// TwinCAT 3 PLC project PRG_B_MachineControl
// Title: B_MachineControl
// Company: RafalOS
// Author: Rafał Osajda
// ProjectVersion: 0.0.0.37
// ProgramVersion: 3.1.4024.0
// libraries:
//   B_Base, * (RafalOS)
//   B_IO, * (RafalOS)
//   B_StatesAndModes, * (RafalOS)
//   Tc2_Standard, * (Beckhoff Automation GmbH)
//   Tc2_System, * (Beckhoff Automation GmbH)
//   Tc3_Module, * (Beckhoff Automation GmbH)
// project tree:
//   / PlcTask.TcTTO (not stored)
//   POUs Compilation/ PRG_Compilation.TcPOU (not stored)
//   POUs/01_MachineControl/ FB_MCMachineControl.TcPOU, ITF_MCMachineControl.TcIO (not stored), ITF_MCMachineControl_HMI_Connector.TcIO, ITF_MCMachineControl_HMI_Init.TcIO, ITF_MCMachineControlConfigure.TcIO, ITF_MCRequiredChange.TcIO (not stored), ST_MCElementListWithParameter.TcDUT, ST_MCRequestChangeMode.TcDUT, ST_MCRequestChangeState.TcDUT (not stored)
//   POUs/02_MachineConfigure/ FB_MCMachineConfigure.TcPOU, ITF_MCConfiguration.TcIO, ITF_MCMachineConfigure.TcIO (not stored)
//   POUs/03_RequiredChange/ FB_MCRequiredChange.TcPOU

// ---- POUs/01_MachineControl/ST_MCElementListWithParameter.TcDUT
TYPE ST_MCElementListWithParameter :
STRUCT
	arrNames 			: ARRAY  [1..GVL_BaseConstans.MAX_NUMBER_OF_ALL_ITEM] OF WSTRING;
	arrID				: ARRAY  [1..GVL_BaseConstans.MAX_NUMBER_OF_ALL_ITEM] OF UINT;
	iNumber				: INT;	//liczba elementów z parametrami
END_STRUCT
END_TYPE

// ---- POUs/01_MachineControl/ST_MCRequestChangeMode.TcDUT
TYPE ST_MCRequestChangeMode :
STRUCT

END_STRUCT
END_TYPE

// ---- POUs/01_MachineControl/ITF_MCMachineControl_HMI_Connector.TcIO
INTERFACE ITF_MCMachineControl_HMI_Connector EXTENDS ITF_BaseTopElement_HMI_Connector

(*			
	RafalOS
	Rafał Osajda		25.11.2025		TC 4024.66
	Zwraca aktualny tryb
*)
METHOD PUBLIC GetActiveMode : E_BaseMachineMode
VAR_INPUT
END_VAR
END_METHOD

METHOD PUBLIC GetActiveModeName : ST_BaseLabel
VAR_INPUT
END_VAR
END_METHOD

(*			
	RafalOS
	Rafał Osajda		25.11.2025		TC 4024.66
	Zwraca aktualny stan
*)
METHOD PUBLIC GetActiveState : E_BaseMachineState
VAR_INPUT
END_VAR
END_METHOD

METHOD PUBLIC GetActiveStateName : ST_BaseLabel
VAR_INPUT
END_VAR
END_METHOD

(*			
	RafalOS
	Rafał Osajda		17.12.2025		TC 4024.66
	Pobiera listę elementów które posiadaja parametr i 
	przypisuje ja do zadanej struktury i zwraca true jak się uda
*)
METHOD GetElementNamesWithParameter : BOOL
VAR_INPUT
	stDane			: REFERENCE TO ST_MCElementListWithParameter;
END_VAR
END_METHOD

METHOD PUBLIC GetModeName : ST_BaseLabel
VAR_INPUT
	iNumber		: INT;
END_VAR
END_METHOD

METHOD PUBLIC GetStateName : ST_BaseLabel
VAR_INPUT
	iNumber		: INT;
END_VAR
END_METHOD

METHOD GetStateTimeForCurrentMode : LTIME
VAR_INPUT
	iNumber			: INT;
END_VAR
END_METHOD

METHOD GetStateTimeForMode : LTIME
VAR_INPUT
	iMode			: INT;
	iState			: INT;
END_VAR
END_METHOD

METHOD PUBLIC GetTimeWorkForMode : LTIME
VAR_INPUT
	iMode	: INT;
END_VAR
END_METHOD

(*			
	RafalOS
	Rafał Osajda		25.11.2025		TC 4024.66
	Zwraca całkowity czas pracy maszyny
*)
METHOD PUBLIC GetTotalWorkTime : LTIME
VAR_INPUT
END_VAR
END_METHOD

(*			
	RafalOS
	Rafał Osajda		25.11.2025		TC 4024.66
	Zwraca czy zmiana trybu sie skoćńzyła
*)
METHOD PUBLIC IsChangeModeDone : BOOL
VAR_INPUT
END_VAR
END_METHOD

(*			
	RafalOS
	Rafał Osajda		25.11.2025		TC 4024.66
	Zwraca czy tryb o podanym numerze jest włączony
*)
METHOD IsModeEnabled : BOOL
VAR_INPUT
	iMode 	: INT;
END_VAR
END_METHOD

(*			
	RafalOS
	Rafał Osajda		24.11.2025		TC 4024.66
	Informacja czy dany stan jest aktywny w aktualnym trybie trybie
*)
METHOD PUBLIC IsStateActiveInCurrentMode : BOOL
VAR_INPUT
END_VAR
END_METHOD

(*			
	RafalOS
	Rafał Osajda		25.11.2025		TC 4024.66
	Informacja czy zadany stan jest stanem aktualnym
*)
METHOD PUBLIC IsStateIsActual : BOOL
VAR_INPUT
	iTestState	: INT;
END_VAR
END_METHOD

METHOD PUBLIC SetCmdChangeMode
VAR_INPUT
	eCmdNumber		: E_SaMCommandChangeMode;
END_VAR
END_METHOD

METHOD PUBLIC SetCmdChangeState
VAR_INPUT
	eCmdNumber		: E_SaMCommandChangeState;
END_VAR
END_METHOD

END_INTERFACE

// ---- POUs/01_MachineControl/ITF_MCMachineControl_HMI_Init.TcIO
INTERFACE ITF_MCMachineControl_HMI_Init EXTENDS ITF_BaseTopElement, ITF_MCMachineControl_HMI_Connector

END_INTERFACE

// ---- POUs/01_MachineControl/ITF_MCMachineControlConfigure.TcIO
(*			
	RafalOS
	Rafał Osajda		29.10.2025		TC 4024.66
	Metody do konfiguracji MAchine control wywoływane z MachineConfigure z pomocą przekazanego ITF
*)
INTERFACE ITF_MCMachineControlConfigure EXTENDS ITF_Base

(*			
	RafalOS
	Rafał Osajda		26.11.2025		TC 4024.66
	Dodawanie szablonu receptury
*)
METHOD PUBLIC AddCreateTemplateFromConfiguration : BOOL
VAR_INPUT
	fbCreateTemplate			: ITF_BaseCreateTemplateOfRecipe;
END_VAR
END_METHOD

(*			
	RafalOS
	Rafał Osajda		13.11.2025		TC 4024.66
	Dodawanie elementów wywoływane z konfiguracji 
*)
METHOD PUBLIC AddElementFromConfiguration : BOOL
VAR_INPUT
	itfElements		: ITF_BaseTopElement;
END_VAR
END_METHOD

(*			
	RafalOS
	Rafał Osajda		13.11.2025		TC 4024.66
	Podpięcie menadżera HMI wywoływane z konfiguracji
*)
METHOD AddHMIManagerFromConfiguration : BOOL
VAR_INPUT
	fbHMIManager			: ITF_BaseGroupElement;
END_VAR
END_METHOD

(*			
	RafalOS
	Rafał Osajda		13.11.2025		TC 4024.66
	Dodanie samego sibie do obsługi w MachineControl
*)
METHOD PUBLIC AddMachineCotrolToYourSelfFromConfiguration : BOOL
VAR_INPUT
END_VAR
END_METHOD

(*			
	RafalOS
	Rafał Osajda		26.11.2025		TC 4024.66
	Dodanie obsługi receptur
*)
METHOD PUBLIC AddModulRecipeFromConfiguration : BOOL
VAR_INPUT
	itfRecipe			: ITF_BaseRecipe;
END_VAR
END_METHOD

(*			
	RafalOS
	Rafał Osajda		13.11.2025		TC 4024.66
	Dodanie modułu sterowania stanami i trybami do machinecontrol z konfiguracji
*)
METHOD PUBLIC AddSaMCotrollerToMachineControlFromConfiguration : BOOL
VAR_INPUT
	itfSaMController			: ITF_SaMController;
END_VAR
END_METHOD

METHOD PUBLIC AddSaMToTopElementFromConfiguration
VAR_INPUT
	itfSaMController			: ITF_SaMController;
END_VAR
END_METHOD

(*			
	RafalOS
	Rafał Osajda		13.11.2025		TC 4024.66
	Wywołanie pierwszego przejścia u wszystkich podzepsołów
*)
METHOD PUBLIC ExecuteFirstCycle : BOOL
VAR_INPUT
END_VAR
END_METHOD

(*			
	RafalOS
	Rafał Osajda		13.11.2025		TC 4024.66
	Zlinkowanie danych wspólnych do dodanych elementów wywoływane z konfiguracji
*)
METHOD PUBLIC LinkCommonDataToAddedElementsFromConfiguration : BOOL
VAR_INPUT
	stCommonData		: REFERENCE TO ST_BaseCommonData;
END_VAR
END_METHOD

(*			
	RafalOS
	Rafał Osajda		13.11.2025		TC 4024.66
	Dodanie głównego komunikatora pomiędzy topelementami do topelementów wywolywane z konfiguracji
*)
METHOD PUBLIC LinkMassangerToaddedTopElementsFromConfiguration : BOOL
VAR_INPUT
	fbCommunicator		: ITF_BaseCommunicator;
END_VAR
END_METHOD

(*			
	RafalOS
	Rafał Osajda		14.11.2025		TC 4024.66
	Podpięcie przyciskow zmiany stanu wywoływane z konfiguracji 
*)
METHOD LinkRequestButtonModeChangeFromConfiguration : BOOL
VAR_INPUT
	iNumberOfRequest			: INT;
	itfRequest					: ITF_MCRequiredChange;
END_VAR
END_METHOD

(*			
	RafalOS
	Rafał Osajda		14.11.2025		TC 4024.66
	Podpięcie przyciskow zmiany trybu i stanu wywoływane z konfiguracji 
*)
METHOD LinkRequestButtonStateChangeFromConfiguration : BOOL
VAR_INPUT
	iNumberOfRequest			: INT;
	itfRequest					: ITF_MCRequiredChange;
END_VAR
END_METHOD

(*			
	RafalOS
	Rafał Osajda		13.11.2025		TC 4024.66
	Podłączenie wsyzstkich zmiennych pochodzących od Programu safety wywoływane w konfiguratorze
*)
METHOD PUBLIC LinkSafetyToaddedElementsFromConfiguration : BOOL
VAR_INPUT
	flSS1				: ITF_BaseFlagGet;
	flSTO				: ITF_BaseFlagGet;
END_VAR
END_METHOD

(*			
	RafalOS
	Rafał Osajda		13.11.2025		TC 4024.66
	Nadanie unikalnych kodów elementom w systemie wywołane z konfiguracji
*)
METHOD PUBLIC SetCodeToAddedElementsFromConfiguration : BOOL
VAR_INPUT
END_VAR
END_METHOD

(*			
	RafalOS
	Rafał Osajda		13.11.2025		TC 4024.66
	Uruchomienie lub wyłączenie obsługi HMI jak jest false fb obsługi nie jest dodawane do MachineControl wywolywane z konfiguracji
*)
METHOD SetEnableHMIServiceFromConfiguration : BOOL
VAR_INPUT
	bValue		: BOOL;
END_VAR
END_METHOD

(*			
	RafalOS
	Rafał Osajda		13.11.2025		TC 4024.66
	Nadaje unikalne ID zgłoszeniom dodanym do elementów w sesyemie wywołane z konfiguracji
*)
METHOD PUBLIC SetIDEventsToAddedElementsFromConfiguration : BOOL
VAR_INPUT
END_VAR
END_METHOD

(*			
	RafalOS
	Rafał Osajda		13.11.2025		TC 4024.66
	Dodanie wszystkim elementom w systemie unikalnego ID
*)
METHOD PUBLIC SetIDToAddedElementsFromConfiguration : BOOL
VAR_INPUT
END_VAR
END_METHOD

(*			
	RafalOS
	Rafał Osajda		14.11.2025		TC 4024.66
	ustawienie trybu poczatkowego wywoływane z konfiguracji
*)
METHOD SetStartModeFromConfiguration : BOOL
VAR_INPUT
	eStartMode				: E_BaseMachineMode;
END_VAR
END_METHOD

END_INTERFACE

// ---- POUs/02_MachineConfigure/ITF_MCConfiguration.TcIO
(*			
	RafalOS
	Rafał Osajda		10.11.2025		TC 4024.66
	Interfejs metod do konfiguracji FB wywoływane z FB_Cofigure
*)
INTERFACE ITF_MCConfiguration

(*			
	RafalOS
	Rafał Osajda		26.11.2025		TC 4024.66
	Dodawanie szablonu receptury
*)
METHOD PUBLIC AddCreateTemplate : BOOL
VAR_INPUT
	itfMachineControl			: ITF_MCMachineControlConfigure;
END_VAR
END_METHOD

(*			
	RafalOS
	Rafał Osajda		13.11.2025		TC 4024.66
	Metoda przeznaczona do dodawania elementów do FB_MachineControl
*)
METHOD PUBLIC AddElements : BOOL
VAR_INPUT
	itfMachineControl			: ITF_MCMachineControlConfigure;
END_VAR
END_METHOD

(*			
	RafalOS
	Rafał Osajda		13.11.2025		TC 4024.66
	Podpięcie menadżera HMI
*)
METHOD AddHMIManager : BOOL
VAR_INPUT
	itfMachineControl			: ITF_MCMachineControlConfigure;
END_VAR
END_METHOD

(*			
	RafalOS
	Rafał Osajda		13.11.2025		TC 4024.66
	Dodanie samego siebie do systemu controli maszyny
*)
METHOD PUBLIC AddMachineCotrolToYourSelf : BOOL
VAR_INPUT
	itfMachineControl			: ITF_MCMachineControlConfigure;
END_VAR
END_METHOD

(*			
	RafalOS
	Rafał Osajda		26.11.2025		TC 4024.66
	Dodanie obsługi receptur
*)
METHOD PUBLIC AddModulRecipe : BOOL
VAR_INPUT
	itfMachineControl			: ITF_MCMachineControlConfigure;
END_VAR
END_METHOD

(*			
	RafalOS
	Rafał Osajda		13.11.2025		TC 4024.66
	Dodanie modułu sterowania stanami i trybami do machinecontrol
*)
METHOD PUBLIC AddSaMCotrollerToMachineControl : BOOL
VAR_INPUT
	itfMachineControl			: ITF_MCMachineControlConfigure;
END_VAR
END_METHOD

METHOD PUBLIC AddSaMToTopElement
VAR_INPUT
	itfMachineControl			: ITF_MCMachineControlConfigure;
END_VAR
END_METHOD

(*			
	RafalOS
	Rafał Osajda		13.11.2025		TC 4024.66
	Zlinkowanie danych wspólnych do dodanych elementów
*)
METHOD PUBLIC LinkCommonDataToAddedElements : BOOL
VAR_INPUT
	itfMachineControl			: ITF_MCMachineControlConfigure;
END_VAR
END_METHOD

(*			
	RafalOS
	Rafał Osajda		13.11.2025		TC 4024.66
	Dodanie głównego komunikatora pomiędzy topelementami do topelementów
*)
METHOD PUBLIC LinkMassangerToaddedTopElements : BOOL
VAR_INPUT
	itfMachineControl			: ITF_MCMachineControlConfigure;
END_VAR
END_METHOD

(*			
	RafalOS
	Rafał Osajda		14.11.2025		TC 4024.66
	Podpięcie przyciskow zmiany trybu i stanu
*)
METHOD LinkRequestButtonChange : BOOL
VAR_INPUT
	itfMachineControl			: ITF_MCMachineControlConfigure;
END_VAR
END_METHOD

(*			
	RafalOS
	Rafał Osajda		13.11.2025		TC 4024.66
	Podłączenie wsyzstkich zmiennych pochodzących od Programu safety 
*)
METHOD PUBLIC LinkSafetyToaddedElements : BOOL
VAR_INPUT
	itfMachineControl			: ITF_MCMachineControlConfigure;
END_VAR
END_METHOD

(*			
	RafalOS
	Rafał Osajda		13.11.2025		TC 4024.66
	Nadanie unikalnych kodów elementom w systemie
*)
METHOD PUBLIC SetCodeToAddedElements : BOOL
VAR_INPUT
	itfMachineControl			: ITF_MCMachineControlConfigure;
END_VAR
END_METHOD

(*			
	RafalOS
	Rafał Osajda		13.11.2025		TC 4024.66
	Uruchomienie lub wyłączenie obsługi HMI jak jest false fb obsługi nie jest dodawane do MachineControl
*)
METHOD SetEnableHMIService : BOOL
VAR_INPUT
	itfMachineControl			: ITF_MCMachineControlConfigure;
END_VAR
END_METHOD

(*			
	RafalOS
	Rafał Osajda		13.11.2025		TC 4024.66
	Nadaje unikalne ID zgłoszeniom dodanym do elementów w sesyemie
*)
METHOD PUBLIC SetIDEventsToAddedElements : BOOL
VAR_INPUT
	itfMachineControl			: ITF_MCMachineControlConfigure;
END_VAR
END_METHOD

(*			
	RafalOS
	Rafał Osajda		13.11.2025		TC 4024.66
	Dodanie wszystkim elementom w systemie unikalnego ID
*)
METHOD PUBLIC SetIDToAddedElements : BOOL
VAR_INPUT
	itfMachineControl			: ITF_MCMachineControlConfigure;
END_VAR
END_METHOD

(*			
	RafalOS
	Rafał Osajda		14.11.2025		TC 4024.66
	ustawienie trybu poczatkowego
*)
METHOD SetStartMode : BOOL
VAR_INPUT
	itfMachineControl			: ITF_MCMachineControlConfigure;
END_VAR
END_METHOD

END_INTERFACE

// ---- POUs/01_MachineControl/FB_MCMachineControl.TcPOU
(*			
	RafalOS
	Rafał Osajda		04.11.2025		TC 4024.66
	Główny FB zarządzający pracą maszyny
*)
FUNCTION_BLOCK FB_MCMachineControl EXTENDS FB_BaseTopElement IMPLEMENTS ITF_MCMachineControl, ITF_MCMachineControlConfigure, ITF_MCMachineControl_HMI_Init
VAR
	(*	Inicjalizacja		*)
	bInitializeCycle			: BOOL;
	bInitDone					: BOOL;
	(*	Konfiguracja		*)
	itfMachineConfigure			: ITF_MCMachineConfigure;		//moduł konfiguracji
	bEnableHMIService			: BOOL;
	(*	TopElementy systemu	*)
	arrTopElements					: ARRAY [1..GVL_BaseConstans.MAX_NUMBER_OF_TOP_ELEMENT] OF ITF_BaseTopElement;
	uiNumberOfAddedTopElement		: UINT := 0;//przy dodawaniu element 0 to system 
	uiNumberOfAllAddedElements		: UINT;		//liczba elementow które są na maszynie 
	(*	Master komunikatora dla top elementów maszyny	*)
	fbMasterCommunicator			: FB_BaseCommunicator;
	(*	Zarządzenia stanami i trybami pracy	*)
	itfSaMController				: ITF_SaMController;
	(*	Stany i Tryby	*)
	arrRequestChangeState			: ARRAY [1..GVL_SaMConstans.NUMBER_OF_COMMAND_CHANGE_STATES] OF ITF_MCRequiredChange;
	arrRequestChangeMode			: ARRAY [1..GVL_SaMConstans.NUMBER_OF_COMMAND_CHANGE_MODES] OF ITF_MCRequiredChange;
	(*	Tablica informacyjna czy praca w stanie aktywnym zakończona	*)
	arrTopElementWorkFinishedInState	: ARRAY [1..GVL_SaMConstans.NUMBER_OF_STATES] OF BOOL;
	(*	Receptury	*)
	itfRecipe						: ITF_BaseRecipe;
	bWorkWithRecipe					: BOOL;
END_VAR
VAR PERSISTENT
	ltWorkTime						: LTIME;				//czas pracy w danym stanie - trybie
END_VAR

IF (NOT THIS^.bInitializeCycle) THEN
	THIS^.bInitializeCycle		:= TRUE;
	THIS^.bInitDone				:= THIS^.InitializeCycle ();
ELSIF (THIS^.bInitDone) THEN
	THIS^.ExecuteCycle ();
END_IF

(*			
	RafalOS
	Rafał Osajda		26.11.2025		TC 4024.66
	Dodawanie szablonu receptury
*)
METHOD PUBLIC AddCreateTemplateFromConfiguration : BOOL
VAR_INPUT
	fbCreateTemplate			: ITF_BaseCreateTemplateOfRecipe;
END_VAR
THIS^.itfRecipe.AddITFToCreateTemplate (fbToCtreateTemplate := fbCreateTemplate);
END_METHOD

(*			
	RafalOS
	Rafał Osajda		13.11.2025		TC 4024.66
	Dodawanie elementów wywoływane z konfiguracji 
*)
METHOD PUBLIC AddElementFromConfiguration : BOOL
VAR_INPUT
	itfElements		: ITF_BaseTopElement;
END_VAR
IF (THIS^.uiNumberOfAddedTopElement + 1 <= GVL_BaseConstans.MAX_NUMBER_OF_TOP_ELEMENT) THEN
	THIS^.uiNumberOfAddedTopElement := THIS^.uiNumberOfAddedTopElement + 1;
	THIS^.arrTopElements [THIS^.uiNumberOfAddedTopElement] := itfElements;

	AddElementFromConfiguration := TRUE;
END_IF
END_METHOD

(*			
	RafalOS
	Rafał Osajda		13.11.2025		TC 4024.66
	Podpięcie menadżera HMI wywoływane z konfiguracji
*)
METHOD AddHMIManagerFromConfiguration : BOOL
VAR_INPUT
	fbHMIManager			: ITF_BaseGroupElement;
END_VAR
IF (THIS^.bEnableHMIService) THEN
	THIS^.AddControlElement (itfControlElement := fbHMIManager);
	
END_IF
END_METHOD

(*			
	RafalOS
	Rafał Osajda		13.11.2025		TC 4024.66
	Dodanie samego sibie do obsługi w MachineControl
*)
METHOD PUBLIC AddMachineCotrolToYourSelfFromConfiguration : BOOL
VAR_INPUT
END_VAR
THIS^.uiNumberOfAddedTopElement := THIS^.uiNumberOfAddedTopElement + 1;
THIS^.arrTopElements [THIS^.uiNumberOfAddedTopElement]	:= THIS^;
END_METHOD

(*			
	RafalOS
	Rafał Osajda		29.10.2025		TC 4024.66
	Dodawanie intefejsu konfiguracji
*)
METHOD PUBLIC AddModulConfigure : BOOL
VAR_INPUT
	fbMachineConfigure			: ITF_MCMachineConfigure;
END_VAR
THIS^.itfMachineConfigure		:= fbMachineConfigure;
END_METHOD

(*			
	RafalOS
	Rafał Osajda		26.11.2025		TC 4024.66
	Dodanie obsługi receptur
*)
METHOD PUBLIC AddModulRecipeFromConfiguration : BOOL
VAR_INPUT
	itfRecipe			: ITF_BaseRecipe;
END_VAR
THIS^.itfRecipe := itfRecipe;
END_METHOD

METHOD PUBLIC AddModulSaM : BOOL
VAR_INPUT
	fbSaMController			: ITF_SaMController;
END_VAR
THIS^.itfSaMController		:= fbSaMController;
THIS^.AddControlElement (itfControlElement	:= fbSaMController);
END_METHOD

(*			
	RafalOS
	Rafał Osajda		13.11.2025		TC 4024.66
	Dodanie modułu sterowania stanami i trybami do machinecontrol z konfiguracji
*)
METHOD PUBLIC AddSaMCotrollerToMachineControlFromConfiguration : BOOL
VAR_INPUT
	itfSaMController			: ITF_SaMController;
END_VAR
VAR
	iNumberOfTopElement			: INT;
END_VAR
THIS^.AddControlElement (itfControlElement := itfSaMController);
THIS^.itfSaMController := itfSaMController;
//FOR iNumberOfTopElement := 1 TO TO_INT (THIS^.uiNumberOfAddedTopElement) DO
//	THIS^.arrTopElements [iNumberOfTopElement].LinkSaM (
//		fbSAM := itfSaMController
//	);
//END_FOR
END_METHOD

METHOD PUBLIC AddSaMToTopElementFromConfiguration
VAR_INPUT
	itfSaMController			: ITF_SaMController;
END_VAR

VAR
	iNumberOfTopElement: INT;
END_VAR
FOR iNumberOfTopElement := 1 TO TO_INT (THIS^.uiNumberOfAddedTopElement) DO
	THIS^.arrTopElements [iNumberOfTopElement].LinkSaM (
		fbSAM := itfSaMController
	);
END_FOR
END_METHOD

METHOD PRIVATE ExecuteCycle
VAR_INST
	tonInterval	: TON;
END_VAR
VAR
	iI			: INT;
	tInterval	: TIME := T#100MS;
END_VAR
	(*	Zarządzanie Stanami i Trybami	*)

THIS^.ExecuteCycle_SaM ();

	(*	Obsługa czasu *)

tonInterval (IN := NOT tonInterval.Q, PT := tInterval);
IF (tonInterval.Q) THEN
	THIS^.itfSaMController.IncrementTimeStateAndMode (tInterval := tInterval);
	THIS^.ltWorkTime := THIS^.ltWorkTime + TO_LTIME (tInterval);
END_IF

	(*	Wywołanie metod obsługiwanych co cykl dla każdego elementu	*)

FOR iI := 1 TO TO_INT (THIS^.uiNumberOfAddedTopElement) DO
	THIS^.arrTopElements [iI].ExecuteEveryCycle_Test ();
	THIS^.arrTopElements [iI].ExecuteEveryCycle_Operation ();
	THIS^.arrTopElements [iI].ExecuteEveryCycle_Status ();
	THIS^.arrTopElements [iI].ExecuteEveryCycle_Error ();
	
END_FOR
END_METHOD

METHOD PRIVATE ExecuteCycle_SaM
VAR
	iI					: INT;
	bBlockade			: BOOL;	//polecenie zmiany trybu i nie sprawdzaj czy jest polecenie zmiany stanu
	bTypeStateActive		: BOOL;
	bTopElementStateWorkCompleted	: BOOL;	//praca w trybach aktywnych zakończona
	
END_VAR

	(*	Zarządzanie stanami i trybami pracy 	*)

IF (NOT THIS^.itfSaMController.IsChangeModeBusy () AND NOT THIS^.itfSaMController.IsChangeStateBusy ()) THEN	
	(*	Testowanie czy jest rządzanie zmiany trybu	*)
	FOR iI := 1 TO GVL_SaMConstans.NUMBER_OF_COMMAND_CHANGE_MODES DO 
		IF (THIS^.arrRequestChangeMode [iI] <> 0) THEN
			IF (THIS^.arrRequestChangeMode [iI].Testing ()) THEN
				THIS^.itfSaMController.Execute (iNumberOfCommand := iI, eChangeCategory := E_SaMChangeCategory.eMode);
				bBlockade		:= TRUE;
				EXIT;
			END_IF
		END_IF
	END_FOR	
	
	(*	Testowanie czy jest rządanie zmiany stany	*)
	IF (NOT bBlockade) THEN
		IF (THIS^.itfSaMController.GetMode () <> E_BaseMachineMode.NotAllowed AND
			THIS^.itfSaMController.GetState () = E_BaseMachineState.Undefined) THEN
			
			THIS^.itfSaMController.Execute (
				iNumberOfCommand := E_SaMCommandChangeState.Abort,
				eChangeCategory := E_SaMChangeCategory.eState
			);
			
		ELSE
			
			FOR iI := 1 TO GVL_SaMConstans.NUMBER_OF_COMMAND_CHANGE_STATES DO 
				IF (THIS^.arrRequestChangeState [iI] <> 0) THEN
					IF (THIS^.arrRequestChangeState [iI].Testing ()) THEN
						THIS^.itfSaMController.Execute (
							iNumberOfCommand := iI,
							eChangeCategory := E_SaMChangeCategory.eState
						);
						EXIT;
					END_IF
				END_IF
			END_FOR
			
		END_IF
	END_IF

END_IF

	(*	Obsługa stanów 		*)
//informacja czy jesteśny w stanie aktywnym	
bTypeStateActive	 := SEL (THIS^.itfSaMController.GetState () <> E_BaseMachineState.Undefined,FALSE,THIS^.itfSaMController.IsStateTypeActive ());
IF (THIS^.itfSaMController.IsChangeModeDone () AND THIS^.itfSaMController.IsChangeStateDone ()) THEN
	bTopElementStateWorkCompleted := bTypeStateActive;
	IF (THIS^.itfSaMController.GetState () <> E_BaseMachineState.Undefined) THEN
		FOR iI := 1 TO TO_INT (THIS^.uiNumberOfAddedTopElement) DO
			IF ( (bTypeStateActive AND NOT THIS^.arrTopElementWorkFinishedInState [iI]) OR NOT bTypeStateActive) THEN
				THIS^.arrTopElementWorkFinishedInState [iI]	:= THIS^.itfSaMController.ExecuteTopElementOperationsForCurrentState (itfTopElement := THIS^.arrTopElements [iI]);
				bTopElementStateWorkCompleted			:= bTopElementStateWorkCompleted AND THIS^.arrTopElementWorkFinishedInState [iI];
			END_IF
		END_FOR
	END_IF
END_IF
(*	OPeracja zakonczona wyczysc tablice dla kolejnej zmiany stanow i konczenia pracy	*)
IF (bTopElementStateWorkCompleted) THEN
	MEMSET (
		destAddr							:= ADR (THIS^.arrTopElementWorkFinishedInState),
		fillByte							:= 0,
		n									:= SIZEOF (THIS^.arrTopElementWorkFinishedInState)
	);
	(*	Zmiana stanu na następny wyjście ze stanu aktywnego	*)
	THIS^.itfSaMController.ExitActivState ();
END_IF
END_METHOD

(*			
	RafalOS
	Rafał Osajda		13.11.2025		TC 4024.66
	Wywołanie pierwszego przejścia u wszystkich podzepsołów
*)
METHOD PUBLIC ExecuteFirstCycle : BOOL
VAR_INPUT
END_VAR

VAR
	iNumberOfTopElement: INT;
END_VAR
FOR iNumberOfTopElement := 1 TO TO_INT (THIS^.uiNumberOfAddedTopElement) DO
	THIS^.arrTopElements [iNumberOfTopElement].FirstCycle ();
END_FOR
END_METHOD

(*			
	RafalOS
	Rafał Osajda		25.11.2025		TC 4024.66
	Zwraca aktualny tryb
*)
METHOD PUBLIC GetActiveMode : E_BaseMachineMode
VAR_INPUT
END_VAR
GetActiveMode := THIS^.itfSaMController.GetMode ();
END_METHOD

METHOD PUBLIC GetActiveModeName : ST_BaseLabel
VAR_INPUT
END_VAR
GetActiveModeName := THIS^.itfSaMController.GetActiveModeName ();
END_METHOD

(*			
	RafalOS
	Rafał Osajda		25.11.2025		TC 4024.66
	Zwraca aktualny stan
*)
METHOD PUBLIC GetActiveState : E_BaseMachineState
VAR_INPUT
END_VAR
GetActiveState := THIS^.itfSaMController.GetState ();
END_METHOD

METHOD PUBLIC GetActiveStateName : ST_BaseLabel
VAR_INPUT
END_VAR
GetActiveStateName := THIS^.itfSaMController.GetActiveStateName ();
END_METHOD

METHOD PUBLIC GetCommunicatorITF : ITF_BaseCommunicator
VAR_INPUT
END_VAR
GetCommunicatorITF := THIS^.fbMasterCommunicator;
END_METHOD

(*			
	RafalOS
	Rafał Osajda		17.12.2025		TC 4024.66
	Pobiera listę elementów które posiadaja parametr i 
	przypisuje ja do zadanej struktury i zwraca true jak się uda
*)
METHOD GetElementNamesWithParameter : BOOL
VAR_INPUT
	stDane			: REFERENCE TO ST_MCElementListWithParameter;
END_VAR

VAR
	iI: INT;
END_VAR
FOR iI := 1 TO TO_INT (THIS^.uiNumberOfAddedTopElement) DO
	;
END_FOR
END_METHOD

METHOD PUBLIC GetModeName : ST_BaseLabel
VAR_INPUT
	iNumber		: INT;
END_VAR
GetModeName := THIS^.itfSaMController.GetModeName (iNumber := iNumber);
END_METHOD

METHOD PUBLIC GetStateName : ST_BaseLabel
VAR_INPUT
	iNumber		: INT;
END_VAR
GetStateName := THIS^.itfSaMController.GetStateName (iNumber := iNumber);
END_METHOD

METHOD GetStateTimeForCurrentMode : LTIME
VAR_INPUT
	iNumber			: INT;
END_VAR
GetStateTimeForCurrentMode := THIS^.itfSaMController. GetTimeStateForCurrentMode (iNumber := iNumber);
END_METHOD

METHOD GetStateTimeForMode : LTIME
VAR_INPUT
	iMode			: INT;
	iState			: INT;
END_VAR
GetStateTimeForMode := THIS^.itfSaMController.GetTimeStateForMode (iMode := iMode, iState := iState);
END_METHOD

(*			
	RafalOS
	Rafał Osajda		25.11.2025		TC 4024.66
	Zrwaca wartośc pracy w trybie
*)
METHOD PUBLIC GetTimeWorkForMode : LTIME
VAR_INPUT
	iMode 	: INT;
END_VAR
GetTimeWorkForMode := THIS^.itfSaMController.GetTimeWorkForMode (iMode := iMode);
END_METHOD

(*			
	RafalOS
	Rafał Osajda		25.11.2025		TC 4024.66
	Zwraca całkowity czas pracy maszyny
*)
METHOD PUBLIC GetTotalWorkTime : LTIME
VAR_INPUT
END_VAR
GetTotalWorkTime := THIS^.ltWorkTime;
END_METHOD

METHOD PRIVATE InitializeCycle : BOOL
VAR
	bResult					: BOOL;
	iI: INT;
END_VAR
bResult				:= TRUE;

bResult				:= bResult AND THIS^.itfMachineConfigure.Configure (fbMachineControl := THIS^);

	(*	Utworzenie szablownów	*)
IF (THIS^.itfRecipe.GetNumberOfTemplate () = 0 OR 
	THIS^.itfRecipe.GetNumberOfCreatingRecipe () <> THIS^.itfRecipe.GetNumberOfTemplate ()
	) THEN
	THIS^.itfRecipe.CreateTemplates ();
	THIS^.bWorkWithRecipe := TRUE;
END_IF

InitializeCycle		:= bResult;
END_METHOD

(*			
	RafalOS
	Rafał Osajda		25.11.2025		TC 4024.66
	Zwraca czy zmiana trybu sie skoćńzyła
*)
METHOD PUBLIC IsChangeModeDone : BOOL
VAR_INPUT
END_VAR
IsChangeModeDone := THIS^.itfSaMController.IsChangeModeDone ();
END_METHOD

METHOD PUBLIC IsInitDone : BOOL
VAR_INPUT
END_VAR
IsInitDone		:= THIS^.bInitDone;
END_METHOD

(*			
	RafalOS
	Rafał Osajda		25.11.2025		TC 4024.66
	Zwraca czy tryb o podanym numerze jest włączony
*)
METHOD IsModeEnabled : BOOL
VAR_INPUT
	iMode 	: INT;
END_VAR
IsModeEnabled := THIS^.itfSaMController.IsModeEnabled (iMode := iMode);
END_METHOD

(*			
	RafalOS
	Rafał Osajda		24.11.2025		TC 4024.66
	Informacja czy dany stan jest aktywny w aktualnym trybie trybie
*)
METHOD PUBLIC IsStateActiveInCurrentMode : BOOL
VAR_INPUT
END_VAR
IsStateActiveInCurrentMode := THIS^.itfSaMController.IsStateInModeEnabled (eStateIn := THIS^.itfSaMController.GetState ());
END_METHOD

(*			
	RafalOS
	Rafał Osajda		25.11.2025		TC 4024.66
	Informacja czy zadany stan jest stanem aktualnym
*)
METHOD PUBLIC IsStateIsActual : BOOL
VAR_INPUT
	iTestState	: INT;
END_VAR
IsStateIsActual := THIS^.itfSaMController.IsStateIsActual (iTestState := iTestState);
END_METHOD

(*			
	RafalOS
	Rafał Osajda		13.11.2025		TC 4024.66
	Zlinkowanie danych wspólnych do dodanych elementów wywoływane z konfiguracji
*)
METHOD PUBLIC LinkCommonDataToAddedElementsFromConfiguration : BOOL
VAR_INPUT
	stCommonData		: REFERENCE TO ST_BaseCommonData;
END_VAR

VAR
	iNumberOfTopElement: INT;
END_VAR
FOR iNumberOfTopElement := 1 TO TO_INT (THIS^.uiNumberOfAddedTopElement) DO
	THIS^.arrTopElements [iNumberOfTopElement].LinkCommonData (
		stCommonData := stCommonData
	);
END_FOR
END_METHOD

(*			
	RafalOS
	Rafał Osajda		13.11.2025		TC 4024.66
	Dodanie głównego komunikatora pomiędzy topelementami do topelementów wywolywane z konfiguracji
*)
METHOD PUBLIC LinkMassangerToaddedTopElementsFromConfiguration : BOOL
VAR_INPUT
	fbCommunicator		: ITF_BaseCommunicator;
END_VAR

VAR
	iI: INT;
END_VAR
THIS^.itfCommunicator := fbCommunicator;

FOR iI := 2 TO TO_INT (THIS^.uiNumberOfAddedTopElement) DO
	THIS^.arrTopElements [iI].LinkCommunicator (fbCommunicator := fbCommunicator);
END_FOR
END_METHOD

(*			
	RafalOS
	Rafał Osajda		14.11.2025		TC 4024.66
	Podpięcie przyciskow zmiany stanu wywoływane z konfiguracji 
*)
METHOD LinkRequestButtonModeChangeFromConfiguration : BOOL
VAR_INPUT
	iNumberOfRequest			: INT;
	itfRequest					: ITF_MCRequiredChange;
END_VAR
THIS^.arrRequestChangeMode [iNumberOfRequest]	:= itfRequest;
END_METHOD

(*			
	RafalOS
	Rafał Osajda		14.11.2025		TC 4024.66
	Podpięcie przyciskow zmiany stanu wywoływane z konfiguracji 
*)
METHOD LinkRequestButtonStateChangeFromConfiguration : BOOL
VAR_INPUT
	iNumberOfRequest			: INT;
	itfRequest					: ITF_MCRequiredChange;
END_VAR
THIS^.arrRequestChangeState [iNumberOfRequest]	:= itfRequest;
END_METHOD

(*			
	RafalOS
	Rafał Osajda		13.11.2025		TC 4024.66
	Podłączenie wsyzstkich zmiennych pochodzących od Programu safety wywoływane w konfiguratorze
*)
METHOD PUBLIC LinkSafetyToaddedElementsFromConfiguration : BOOL
VAR_INPUT
	flSS1				: ITF_BaseFlagGet;
	flSTO				: ITF_BaseFlagGet;
END_VAR

VAR
	iI: INT;
END_VAR
THIS^.LinkSS1 (fbSS1 := flSS1);
THIS^.LinkSTO (fbSTO := flSTO);

FOR iI := 2 TO TO_INT (THIS^.uiNumberOfAddedTopElement) DO
	THIS^.arrTopElements [iI].LinkSS1 (fbSS1 := flSS1);
	THIS^.arrTopElements [iI].LinkSTO (fbSTO := flSTO);
END_FOR
END_METHOD

METHOD PUBLIC SetCmdChangeMode
VAR_INPUT
	eCmdNumber		: E_SaMCommandChangeMode;
END_VAR
THIS^.arrRequestChangeMode [eCmdNumber].SetRequiredChange (bIn := TRUE);
END_METHOD

METHOD PUBLIC SetCmdChangeState
VAR_INPUT
	eCmdNumber		: E_SaMCommandChangeState;
END_VAR
THIS^.arrRequestChangeState [eCmdNumber].SetRequiredChange (bIn := TRUE);
END_METHOD

(*			
	RafalOS
	Rafał Osajda		13.11.2025		TC 4024.66
	Nadanie unikalnych kodów elementom w systemie wywołane z konfiguracji
*)
METHOD PUBLIC SetCodeToAddedElementsFromConfiguration : BOOL
VAR_INPUT
END_VAR

VAR
	iNumberOfTopElement: INT;
END_VAR
FOR iNumberOfTopElement := 1 TO TO_INT (THIS^.uiNumberOfAddedTopElement) DO
	THIS^.arrTopElements [iNumberOfTopElement].SetCode (
		sCode := '0.0.0.0.0', sAdd := TO_STRING (iNumberOfTopElement)
	);
END_FOR
END_METHOD

(*			
	RafalOS
	Rafał Osajda		13.11.2025		TC 4024.66
	Uruchomienie lub wyłączenie obsługi HMI jak jest false fb obsługi nie jest dodawane do MachineControl wywolywane z konfiguracji
*)
METHOD SetEnableHMIServiceFromConfiguration : BOOL
VAR_INPUT
	bValue		: BOOL;
END_VAR
THIS^.bEnableHMIService := bValue;
END_METHOD

(*			
	RafalOS
	Rafał Osajda		13.11.2025		TC 4024.66
	Nadaje unikalne ID zgłoszeniom dodanym do elementów w sesyemie wywołane z konfiguracji
*)
METHOD PUBLIC SetIDEventsToAddedElementsFromConfiguration : BOOL
VAR_INPUT
END_VAR
VAR
	iNumberOfTopElement	: INT;
END_VAR
FOR iNumberOfTopElement := 1 TO TO_INT (THIS^.uiNumberOfAddedTopElement) DO
	THIS^.refstCommonData.itfLogger.SetNumerOfReportsIntheSystem (
			uiValue := THIS^.arrTopElements [iNumberOfTopElement].SetEventsIDs (
				uiNewID := THIS^.refstCommonData.itfLogger.GetNumerOfReportsIntheSystem ()
			)
	);
END_FOR
END_METHOD

(*			
	RafalOS
	Rafał Osajda		13.11.2025		TC 4024.66
	Dodanie wszystkim elementom w systemie unikalnego ID
*)
METHOD PUBLIC SetIDToAddedElementsFromConfiguration : BOOL
VAR_INPUT
END_VAR
VAR
	iNumberOfTopElement		: INT;
END_VAR
FOR iNumberOfTopElement := 1 TO TO_INT (THIS^.uiNumberOfAddedTopElement) DO
	THIS^.uiNumberOfAllAddedElements := 
		THIS^.arrTopElements [iNumberOfTopElement].SetID (
			uiID := THIS^.uiNumberOfAllAddedElements + 1
		);
END_FOR
END_METHOD

(*			
	RafalOS
	Rafał Osajda		14.11.2025		TC 4024.66
	ustawienie trybu poczatkowego wywoływane z konfiguracji
*)
METHOD SetStartModeFromConfiguration : BOOL
VAR_INPUT
	eStartMode				: E_BaseMachineMode;
END_VAR
THIS^.itfSaMController.Execute (iNumberOfCommand := eStartMode, eChangeCategory := E_SaMChangeCategory.eMode);
END_METHOD

METHOD STARE_AddHMIManager : BOOL
VAR_INPUT
	itfHMIManager			: ITF_BaseGroupElement;
END_VAR
THIS^.AddControlElement (itfControlElement := itfHMIManager);
END_METHOD

(*			
	RafalOS
	Rafał Osajda		29.10.2025		TC 4024.66
	Metoda dodawania top elementu wywoływana z konfiguracji
*)
METHOD STARE_AddTopElementFromConfiguration : BOOL
VAR_INPUT
	fbTopElement		: ITF_BaseTopElement;
END_VAR
IF (THIS^.uiNumberOfAddedTopElement + 1 <= GVL_BaseConstans.MAX_NUMBER_OF_TOP_ELEMENT) THEN
	THIS^.uiNumberOfAddedTopElement							:= THIS^.uiNumberOfAddedTopElement + 1;
	THIS^.arrTopElements [THIS^.uiNumberOfAddedTopElement]	:= fbTopElement;
	
	THIS^.arrTopElements [THIS^.uiNumberOfAddedTopElement].LinkCommonData (stCommonData	:= THIS^.refstCommonData);
	THIS^.arrTopElements [THIS^.uiNumberOfAddedTopElement].LinkSS1 (fbSS1	:= THIS^.itfSS1);
	THIS^.arrTopElements [THIS^.uiNumberOfAddedTopElement].LinkSTO (fbSTO	:= THIS^.itfSTO);
	THIS^.arrTopElements [THIS^.uiNumberOfAddedTopElement].LinkCommunicator (fbCommunicator	:= THIS^.fbMasterCommunicator);
	(*	Podpięcie systemu sterowania stanami i trybami	*)
	THIS^.arrTopElements [THIS^.uiNumberOfAddedTopElement].LinkSAM (fbSAM	:= THIS^.itfSaMController);
	THIS^.arrTopElements [THIS^.uiNumberOfAddedTopElement].FirstCycle ();
	THIS^.uiNumberOfAllAddedElements 						:= THIS^.arrTopElements [THIS^.uiNumberOfAddedTopElement].SetID (uiID := THIS^.uiNumberOfAllAddedElements + 1);
	THIS^.refstCommonData.itfLogger.SetNumerOfReportsIntheSystem (
			uiValue := THIS^.arrTopElements [THIS^.uiNumberOfAddedTopElement].SetEventsIDs (
				uiNewID := THIS^.refstCommonData.itfLogger.GetNumerOfReportsIntheSystem ()
			)
	);
	THIS^.arrTopElements [THIS^.uiNumberOfAddedTopElement].SetCode (sCode := '0.0.0.0.0', sAdd := TO_STRING (THIS^.uiNumberOfAddedTopElement));
	
	STARE_AddTopElementFromConfiguration							:= TRUE;
END_IF
END_METHOD

END_FUNCTION_BLOCK

// ---- POUs/02_MachineConfigure/FB_MCMachineConfigure.TcPOU
FUNCTION_BLOCK FB_MCMachineConfigure EXTENDS FB_Base IMPLEMENTS ITF_MCMachineConfigure
VAR
	(*	Baza konfiguracji	*)
	arritfConfigure				: ARRAY [1..10] OF ITF_MCConfiguration;
	iNubmerOfAddedConfigure		: INT;
END_VAR

METHOD PUBLIC AddConfiguration : BOOL
VAR_INPUT
	fbConfigure		: ITF_MCConfiguration;
END_VAR
IF (THIS^.iNubmerOfAddedConfigure + 1 <= 10) THEN
	THIS^.iNubmerOfAddedConfigure	:= THIS^.iNubmerOfAddedConfigure + 1;
	THIS^.arritfConfigure [THIS^.iNubmerOfAddedConfigure]	:= fbConfigure;
	AddConfiguration	:= TRUE;
ELSE
	AddConfiguration	:= FALSE;
END_IF
END_METHOD

METHOD PUBLIC Configure : BOOL
VAR_INPUT
	fbMachineControl	: ITF_MCMachineControlConfigure;
END_VAR

VAR
	bResult				: BOOL;
	iI					: INT;
END_VAR
bResult			:= TRUE;

THIS^.arritfConfigure [1].AddMachineCotrolToYourSelf (itfMachineControl := fbMachineControl);
THIS^.arritfConfigure [1].AddSaMCotrollerToMachineControl (itfMachineControl := fbMachineControl);
THIS^.arritfConfigure [1].AddModulRecipe (itfMachineControl := fbMachineControl);
FOR iI := 1 TO THIS^.iNubmerOfAddedConfigure DO 
	IF (THIS^.arritfConfigure [iI] <> 0) THEN
		
		THIS^.arritfConfigure [iI].SetEnableHMIService (itfMachineControl := fbMachineControl);
		THIS^.arritfConfigure [iI].AddHMIManager (itfMachineControl := fbMachineControl);
		THIS^.arritfConfigure [iI].AddElements (itfMachineControl	:= fbMachineControl);
		THIS^.arritfConfigure [iI].LinkRequestButtonChange (itfMachineControl	:= fbMachineControl);
		THIS^.arritfConfigure [iI].SetStartMode (itfMachineControl	:= fbMachineControl);
		THIS^.arritfConfigure [iI].AddCreateTemplate (itfMachineControl	:= fbMachineControl);
	END_IF
END_FOR



THIS^.arritfConfigure [1].LinkCommonDataToAddedElements (itfMachineControl := fbMachineControl);
THIS^.arritfConfigure [1].SetIDToAddedElements (itfMachineControl := fbMachineControl);
fbMachineControl.ExecuteFirstCycle ();
THIS^.arritfConfigure [1].SetIDEventsToAddedElements (itfMachineControl := fbMachineControl);
THIS^.arritfConfigure [1].SetCodeToAddedElements (itfMachineControl := fbMachineControl);
THIS^.arritfConfigure [1].LinkSafetyToAddedElements (itfMachineControl := fbMachineControl);
THIS^.arritfConfigure [1].AddSaMToTopElement (itfMachineControl := fbMachineControl);
THIS^.arritfConfigure [1].LinkMassangerToaddedTopElements (itfMachineControl := fbMachineControl);

Configure		:= bResult;
END_METHOD

END_FUNCTION_BLOCK

// ---- POUs/03_RequiredChange/FB_MCRequiredChange.TcPOU
(*			
	RafalOS
	Rafał Osajda		04.11.2025		TC 4024.66
	Polecenie zmiany trybu lub stanu - rozszerzony przycisk o możliwość sterowania z HMI i na wyjściu daje mi impuls na jeden cykl
*)
FUNCTION_BLOCK FB_MCRequiredChange EXTENDS FB_IOButton_NO IMPLEMENTS ITF_MCRequiredChange
VAR
	bChange					: BOOL;
	rtChange				: Tc2_Standard.R_TRIG;
END_VAR

METHOD PUBLIC SetRequiredChange
VAR_INPUT
	bIn: BOOL;
END_VAR
THIS^.bChange		:= bIn;
END_METHOD

(*			
	RafalOS
	Rafał Osajda		04.11.2025		TC 4024.66
	
*)
METHOD Testing : BOOL
VAR_INPUT
END_VAR
THIS^.rtChange (CLK	:= THIS^.IsPressed () OR THIS^.bChange);
THIS^.bChange	:= FALSE;
Testing			:= THIS^.rtChange.Q;
END_METHOD

END_FUNCTION_BLOCK
